// Alias for error code.
TYPE T_ErrorCode : LINT; END_TYPE

(* stored: Version 1.1.0.1
   DUT T_ErrorCode: Id {b70c1957-df68-0090-1cc5-1b4104a869c2} *)
